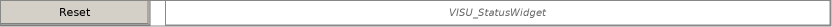
VISUALIZATION VISU_Axes_Commands_Reset  // 832x27
VAR_IN_OUT
    reset : Process;
    resetStatus : StatusWidget;
END_VAR
    Button (0,0 150x25), "Reset", input disabled if: reset.statuses.enabledStatus.disabled
        OnMouseClick: execute { reset.request(); }
    Frame (165,0 665x25)
        shows VISU_StatusWidget(widget := resetStatus)
END_VISUALIZATION

(* stored: Version 1.1.0.1, ProductVersion 3.1.4019.2
   Visu VISU_Axes_Commands_Reset: Id {67ac0106-bb1e-41ff-97e6-e2f5e475b365} *)
